(* CODESYS project CodesysElevator.project

Project tree, tasks and I/O mapping:
  CODESYS_Control_Win_V3_x64 : CODESYS Control Win V3 x64, 3S - Smart Software Solutions GmbH, version 3.5.12.30
    application Application
      libraries: BASIC, 3.31 (OSCAT); Util, * (System)
      task VISU_TASK (cyclic, interval 50 ms, priority 31) calls VisuElems.Visu_Prg
      task Task (cyclic, interval t#20ms, priority 1) calls SimulationLogic, main
      Simulation/
        simcomponents/
          visualisation FloorButtons
          visualisation Door
          visualisation Elevator
        SimulationHelpers/
          function block MoveObject [ST]
          function block DoorLogic [ST]
        simlogic/
          program SimIO [ST]
          program SimulationLogic [ST]
        visualisation theLab
      IOs/
        global variables SystemState
        global variables IOs
      control/
        program ElevatorControl [LD]
        program main [ST]
        function block DoorCtrl [SFC]
  libraries: SysTimeCore, 3.5.5.0 (System)
  text list GlobalTextList
*)

// CODESYS_Control_Win_V3_x64/Application/IOs/SystemState
VAR_GLOBAL
	useInputsFromSimulation: BOOL := TRUE;
END_VAR

// CODESYS_Control_Win_V3_x64/Application/IOs/IOs
VAR_GLOBAL
	// inputs
	// Buttons
	ixButtonInElevatorF1: BOOL; // a request in the elevator to go to floor 1
	ixButtonInElevatorF2: BOOL;
	ixButtonInElevatorF3: BOOL;
	ixButtonInElevatorF4: BOOL;
	ixButtonInElevatorCloseDoors: BOOL; // a request to close the door inside the elevator if possible
	ixButtonInElevatorOpenDoors: BOOL; // a request to open the door inside the elevator if possible
	
	// security and sensors
	ixEmergencyStop: BOOL; // Emergency stop is pressed
	ixElevatorAt1: BOOL; // the elevator is at F1 sensor
	ixElevatorAt2: BOOL;
	ixElevatorAt3: BOOL;
	ixElevatorAt4: BOOL;
	ixDoorOpenedF1: BOOL; // the door is fully opened at F1
	ixDoorClosedF1: BOOL; // the door is fully closed at F1
	ixDoorOpenedF2: BOOL;
	ixDoorClosedF2: BOOL;
	ixDoorOpenedF3: BOOL;
	ixDoorClosedF3: BOOL;
	ixDoorOpenedF4: BOOL;
	ixDoorClosedF4: BOOL;

	// outputs
	// lamps
	qxLampInElevatorF1: BOOL;
	qxLampInElevatorF2: BOOL;
	qxLampInElevatorF3: BOOL;
	qxLampInElevatorF4: BOOL;
	qxLampEmergencyStop: BOOL;
	
	qxElevatorGoUp: BOOL;
	qxElevatorGoDown: BOOL;
	qxOpenDoorF1: BOOL; // Opens the door at F1, closes if false
	qxOpenDoorF2: BOOL; // Opens the door at F1, closes if false
	qxOpenDoorF3: BOOL; // Opens the door at F1, closes if false
	qxOpenDoorF4: BOOL; // Opens the door at F1, closes if false
	
END_VAR

// CODESYS_Control_Win_V3_x64/Application/Simulation/simlogic/SimulationLogic
PROGRAM SimulationLogic
VAR
	moveElevator: MoveObject;
	onlyForSimulationElevatorPosY: INT := 0;
	dummyZeroPos: INT := 0;
	elevatorMoving: BOOL;
	
	doorHandleF1: DoorLogic;
	leftPosF1: INT;
	rightPosF1: INT;	
	
	doorHandleF2: DoorLogic;
	leftPosF2: INT;
	rightPosF2: INT;	
	
	doorHandleF3: DoorLogic;
	leftPosF3: INT;
	rightPosF3: INT;	
	
	doorHandleF4: DoorLogic;
	leftPosF4: INT;
	rightPosF4: INT;
	

	
END_VAR


SimIO();



doorHandleF1(leftPos:=leftPosF1, rightPos:= rightPosF1, sensor:= ixElevatorAt1, open := qxOpenDoorF1, close := NOT qxOpenDoorF1);
doorHandleF2(leftPos:=leftPosF2, rightPos:= rightPosF2, sensor:= ixElevatorAt2, open := qxOpenDoorF2, close := NOT qxOpenDoorF2);
doorHandleF3(leftPos:=leftPosF3, rightPos:= rightPosF3, sensor:= ixElevatorAt3, open := qxOpenDoorF3, close := NOT qxOpenDoorF3);
doorHandleF4(leftPos:=leftPosF4, rightPos:= rightPosF4, sensor:= ixElevatorAt4, open := qxOpenDoorF4, close := NOT qxOpenDoorF4);
	

moveElevator(
	moveUP:= SimIO.sim_qxElevatorGoUp, 
	moveDown:= SimIO.sim_qxElevatorGoDown, 
	moveLeft:=FALSE , 
	moveRight:=FALSE , 
	maxX:=0, 
	minX:=0, 
	maxY:=340, 
	minY:=-30, 
	tick:=T#0.03S , 
	x:= dummyZeroPos, 
	y:= onlyForSimulationElevatorPosY );
	
elevatorMoving := moveElevator.isMoving;

END_PROGRAM

// CODESYS_Control_Win_V3_x64/Application/Simulation/simlogic/SimIO
PROGRAM SimIO
VAR
	
	simpleHysteresis: INT := 2;
	posF4: INT := -23;
	posF3: INT := 97;
	posF2: INT := 218;
	posF1: INT := 338;
	
		// for internal simulation use and a way to change bewteen sim and real
	sim_ixButtonAtF1Up: BOOL; 
	sim_ixButtonAtF2Down: BOOL; 
	sim_ixButtonAtF2Up: BOOL;   
	sim_ixButtonAtF3Down: BOOL;
	sim_ixButtonAtF3Up: BOOL;
	sim_ixButtonAtF4Down: BOOL;
	sim_ixButtonInElevatorF1: BOOL; 
	sim_ixButtonInElevatorF2: BOOL;
	sim_ixButtonInElevatorF3: BOOL;
	sim_ixButtonInElevatorF4: BOOL;
	sim_ixButtonInElevatorCloseDoors: BOOL; 
	sim_ixButtonInElevatorOpenDoors: BOOL; 
	
	sim_ixDoorSensorInElevator: BOOL; 
	sim_ixEmergencyStop: BOOL; 
	sim_ixElevatorAt1: BOOL; 
	sim_ixElevatorAt2: BOOL;
	sim_ixElevatorAt3: BOOL;
	sim_ixElevatorAt4: BOOL;
	sim_ixDoorOpenedF1: BOOL; 
	sim_ixDoorClosedF1: BOOL; 
	sim_ixDoorOpenedF2: BOOL;
	sim_ixDoorClosedF2: BOOL;
	sim_ixDoorOpenedF3: BOOL;
	sim_ixDoorClosedF3: BOOL;
	sim_ixDoorOpenedF4: BOOL;
	sim_ixDoorClosedF4: BOOL;

	sim_qxLampAtF1Up: BOOL;
	sim_qxLampAtF2Down: BOOL;
	sim_qxLampAtF2Up: BOOL;
	sim_qxLampAtF3Down: BOOL;
	sim_qxLampAtF3Up: BOOL;
	sim_qxLampAtF4Down: BOOL;
	sim_qxLampInElevatorF1: BOOL;
	sim_qxLampInElevatorF2: BOOL;
	sim_qxLampInElevatorF3: BOOL;
	sim_qxLampInElevatorF4: BOOL;
	sim_qxLampEmergencyStop: BOOL;
	
	sim_qxElevatorGoUp: BOOL;
	sim_qxElevatorGoDown: BOOL;
	sim_qxOpenDoorF1: BOOL; 
	sim_qxOpenDoorF2: BOOL; 
	sim_qxOpenDoorF3: BOOL; 
	sim_qxOpenDoorF4: BOOL; 
END_VAR

// logic

SimIO.sim_ixElevatorAt1 := SimulationLogic.onlyForSimulationElevatorPosY > posF1;
SimIO.sim_ixElevatorAt2 := SimulationLogic.onlyForSimulationElevatorPosY < posF2+simpleHysteresis AND SimulationLogic.onlyForSimulationElevatorPosY > posF2-simpleHysteresis;
SimIO.sim_ixElevatorAt3 := SimulationLogic.onlyForSimulationElevatorPosY < posF3+simpleHysteresis AND SimulationLogic.onlyForSimulationElevatorPosY > posF3-simpleHysteresis;
SimIO.sim_ixElevatorAt4 := SimulationLogic.onlyForSimulationElevatorPosY < posF4;

sim_ixDoorOpenedF1 := SimulationLogic.doorHandleF1.opened;
sim_ixDoorClosedF1 := SimulationLogic.doorHandleF1.closed;
sim_ixDoorOpenedF2 := SimulationLogic.doorHandleF2.opened;
sim_ixDoorClosedF2 := SimulationLogic.doorHandleF2.closed;
sim_ixDoorOpenedF3 := SimulationLogic.doorHandleF3.opened;
sim_ixDoorClosedF3 := SimulationLogic.doorHandleF3.closed;
sim_ixDoorOpenedF4 := SimulationLogic.doorHandleF4.opened;
sim_ixDoorClosedF4 := SimulationLogic.doorHandleF4.closed;


// mapping
IF useInputsFromSimulation THEN
	ixButtonInElevatorF1:=sim_ixButtonInElevatorF1;
	ixButtonInElevatorF2:=sim_ixButtonInElevatorF2;
	ixButtonInElevatorF3:=sim_ixButtonInElevatorF3;
	ixButtonInElevatorF4:=sim_ixButtonInElevatorF4;
	ixButtonInElevatorCloseDoors:=sim_ixButtonInElevatorCloseDoors;
	ixButtonInElevatorOpenDoors:=sim_ixButtonInElevatorOpenDoors;
	
	ixEmergencyStop:=sim_ixEmergencyStop;
	ixElevatorAt1:=sim_ixElevatorAt1;
	ixElevatorAt2:=sim_ixElevatorAt2;
	ixElevatorAt3:=sim_ixElevatorAt3;
	ixElevatorAt4:=sim_ixElevatorAt4;
	ixDoorOpenedF1:=sim_ixDoorOpenedF1;
	ixDoorClosedF1:=sim_ixDoorClosedF1;
	ixDoorOpenedF2:=sim_ixDoorOpenedF2;
	ixDoorClosedF2:=sim_ixDoorClosedF2;
	ixDoorOpenedF3:=sim_ixDoorOpenedF3;
	ixDoorClosedF3:=sim_ixDoorClosedF3;
	ixDoorOpenedF4:=sim_ixDoorOpenedF4;
	ixDoorClosedF4:=sim_ixDoorClosedF4;
END_IF

	sim_qxLampInElevatorF1:=qxLampInElevatorF1;
	sim_qxLampInElevatorF2:=qxLampInElevatorF2;
	sim_qxLampInElevatorF3:=qxLampInElevatorF3;
	sim_qxLampInElevatorF4:=qxLampInElevatorF4;
	sim_qxLampEmergencyStop:=qxLampEmergencyStop;
	
	sim_qxElevatorGoUp:=qxElevatorGoUp;
	sim_qxElevatorGoDown:=qxElevatorGoDown;
	sim_qxOpenDoorF1:=qxOpenDoorF1;
	sim_qxOpenDoorF2:=qxOpenDoorF2;
	sim_qxOpenDoorF3:=qxOpenDoorF3;
	sim_qxOpenDoorF4:=qxOpenDoorF4;

END_PROGRAM

// CODESYS_Control_Win_V3_x64/Application/Simulation/SimulationHelpers/MoveObject
FUNCTION_BLOCK MoveObject
VAR_INPUT
	moveUP: BOOL;
	moveDown: BOOL;
	moveLeft: BOOL;
	moveRight: BOOL;
	maxX: INT;
	minX: INT;
	maxY: INT;
	minY: INT;
	tick: time;
END_VAR
VAR_IN_OUT
	x: INT;
	y: INT;
END_VAR
VAR_OUTPUT
	isMoving: BOOL;
END_VAR
VAR
	pulse: CLK_PULSE;
END_VAR

pulse(
	PT:= tick, 
	N:= 0, 
	RST:= NOT moveUp AND NOT moveDown AND NOT moveLeft AND NOT moveRight , 
	Q=> , 
	CNT=> , 
	RUN=> );
	
IF pulse.Q THEN
	IF moveUP AND NOT moveDown AND y > minY THEN
		y := y-1; 
	ELSIF NOT moveUP AND moveDown AND y < maxY THEN
		y := y+1;
	END_IF
	
	IF moveRight AND NOT moveLeft AND x < maxX THEN
		x := x+1;
	ELSIF NOT moveRight AND moveLeft AND x > minX THEN
		x := x-1;
	END_IF
END_IF

isMoving := moveUP OR moveDown;

END_FUNCTION_BLOCK

// CODESYS_Control_Win_V3_x64/Application/Simulation/SimulationHelpers/DoorLogic
FUNCTION_BLOCK DoorLogic
VAR_INPUT
	open: BOOL;
	close: BOOL;
	sensor: BOOL;
END_VAR
VAR_OUTPUT
	opened: BOOL;
	closed: BOOL;
END_VAR
VAR_IN_OUT
	leftPos: INT;
	rightPos: INT;
END_VAR
VAR
	moveLeft: MoveObject;
	moveRight: MoveObject;
	dummy: INT;
	doOpen: BOOL;
	doClose: BOOL;
END_VAR


opened := leftPos <= -60 AND rightPos >= 60;
closed := leftPos >= 0 AND rightPos <= 0;

doOpen := open AND NOT opened AND NOT close;
doClose := close AND NOT closed AND NOT open;


moveLeft(
	moveUP:= FALSE, 
	moveDown:= FALSE, 
	moveLeft:=doOpen, 
	moveRight:=doClose, 
	maxX:=300, 
	minX:=-300, 
	maxY:=0, 
	minY:=0, 
	tick:=T#0.03S , 
	x:= leftPos, 
	y:= dummy
);

moveRight(
	moveUP:= FALSE, 
	moveDown:= FALSE, 
	moveLeft:=doClose , 
	moveRight:=doOpen , 
	maxX:=300, 
	minX:=-300, 
	maxY:=0, 
	minY:=0, 
	tick:=T#0.03S , 
	x:= rightPos, 
	y:= dummy
);

END_FUNCTION_BLOCK

// CODESYS_Control_Win_V3_x64/Application/control/main
PROGRAM main
VAR
END_VAR

ElevatorControl();

END_PROGRAM

// CODESYS_Control_Win_V3_x64/Application/control/ElevatorControl
PROGRAM ElevatorControl
VAR
	requestF1: BOOL := FALSE;
	requestF2: BOOL := FALSE;
	requestF3: BOOL := FALSE;
	requestF4: BOOL := TRUE;
	r1: BOOL;
	r2: BOOL;
	r3: BOOL;
	r4: BOOL := TRUE;
	up: BOOL := TRUE;
	down: BOOL;
	doorF1: DoorCtrl;
	doorF2: DoorCtrl;
	doorF3: DoorCtrl;
	doorF4: DoorCtrl;
	insane_closing_skills: BOOL := TRUE;
	not_moving: BOOL;
	insane_opening_skills: BOOL;
	going_up: BOOL := TRUE;
	executing1: BOOL;
	executing2: BOOL;
	executing3: BOOL;
	executing4: BOOL;
	executing: BOOL;
	at_stop: BOOL;
	lastF1: BOOL;
	lastF2: BOOL;
	lastF3: BOOL;
	lastF4: BOOL;
END_VAR
VAR // added by the converter: edge detectors and wires of the graphical bodies
    _rt1, _rt2, _rt3, _rt4, _rt5 : R_TRIG;
    _ft1, _ft2, _ft3, _ft4, _ft5, _ft6, _ft7, _ft8, _ft9, _ft10, _ft11, _ft12 : F_TRIG;
END_VAR

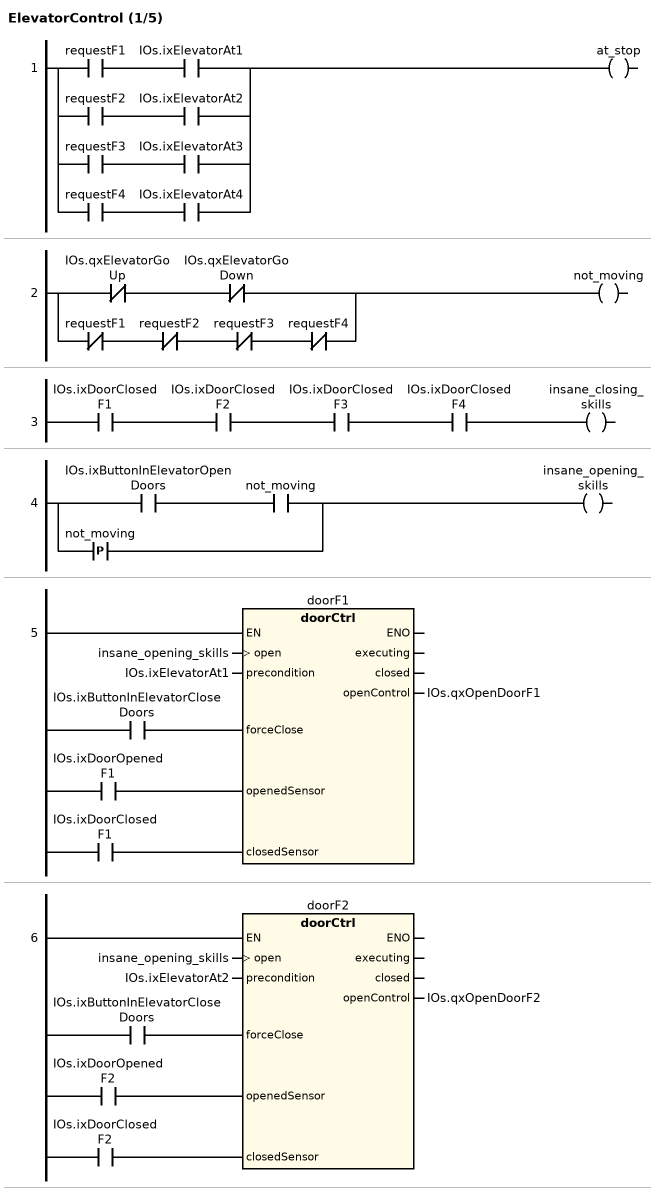
// NETWORK 1
at_stop := requestF1 AND IOs.ixElevatorAt1 OR requestF2 AND IOs.ixElevatorAt2 OR requestF3 AND IOs.ixElevatorAt3 OR requestF4 AND IOs.ixElevatorAt4;

// NETWORK 2
not_moving := NOT IOs.qxElevatorGoUp AND NOT IOs.qxElevatorGoDown OR NOT requestF1 AND NOT requestF2 AND NOT requestF3 AND NOT requestF4;

// NETWORK 3
insane_closing_skills := IOs.ixDoorClosedF1 AND IOs.ixDoorClosedF2 AND IOs.ixDoorClosedF3 AND IOs.ixDoorClosedF4;

// NETWORK 4
_rt1(CLK := not_moving);
insane_opening_skills := IOs.ixButtonInElevatorOpenDoors AND not_moving OR _rt1.Q;

// NETWORK 5
_rt2(CLK := insane_opening_skills);
doorF1(
    open := _rt2.Q,
    precondition := IOs.ixElevatorAt1,
    forceClose := IOs.ixButtonInElevatorCloseDoors,
    openedSensor := IOs.ixDoorOpenedF1,
    closedSensor := IOs.ixDoorClosedF1,
    openControl => IOs.qxOpenDoorF1); // doorCtrl

// NETWORK 6
_rt3(CLK := insane_opening_skills);
doorF2(
    open := _rt3.Q,
    precondition := IOs.ixElevatorAt2,
    forceClose := IOs.ixButtonInElevatorCloseDoors,
    openedSensor := IOs.ixDoorOpenedF2,
    closedSensor := IOs.ixDoorClosedF2,
    openControl => IOs.qxOpenDoorF2); // doorCtrl

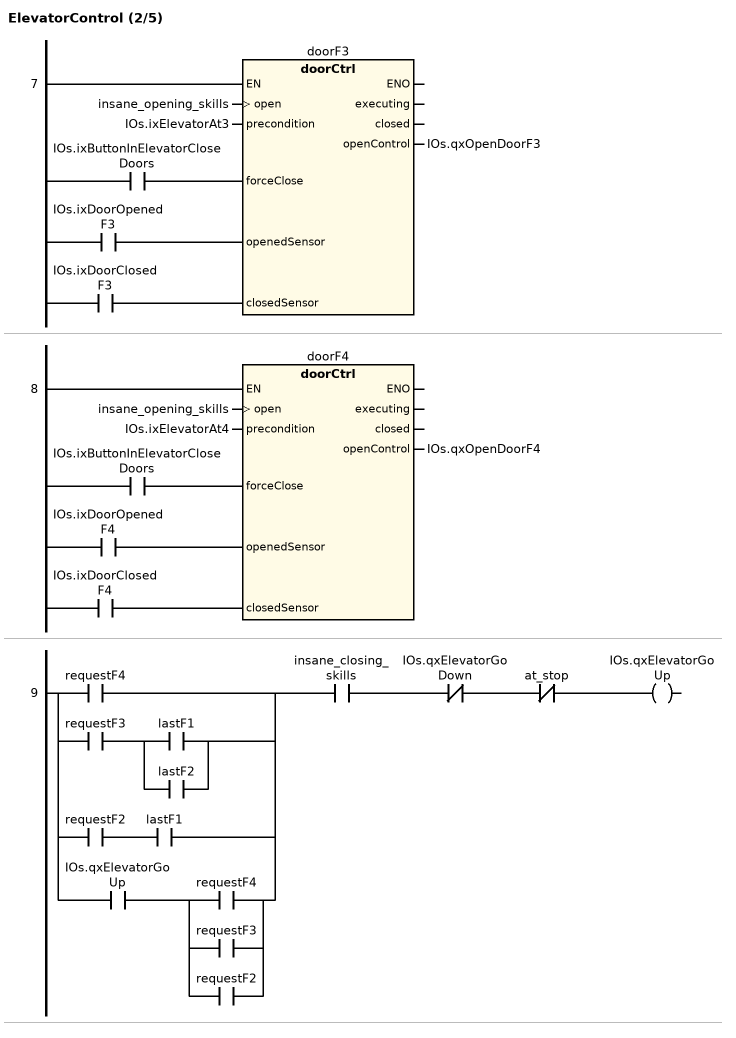
// NETWORK 7
_rt4(CLK := insane_opening_skills);
doorF3(
    open := _rt4.Q,
    precondition := IOs.ixElevatorAt3,
    forceClose := IOs.ixButtonInElevatorCloseDoors,
    openedSensor := IOs.ixDoorOpenedF3,
    closedSensor := IOs.ixDoorClosedF3,
    openControl => IOs.qxOpenDoorF3); // doorCtrl

// NETWORK 8
_rt5(CLK := insane_opening_skills);
doorF4(
    open := _rt5.Q,
    precondition := IOs.ixElevatorAt4,
    forceClose := IOs.ixButtonInElevatorCloseDoors,
    openedSensor := IOs.ixDoorOpenedF4,
    closedSensor := IOs.ixDoorClosedF4,
    openControl => IOs.qxOpenDoorF4); // doorCtrl

// NETWORK 9
IOs.qxElevatorGoUp := (requestF4 OR requestF3 AND (lastF1 OR lastF2) OR requestF2 AND lastF1 OR IOs.qxElevatorGoUp AND (requestF4 OR requestF3 OR requestF2)) AND insane_closing_skills AND NOT IOs.qxElevatorGoDown AND NOT at_stop;

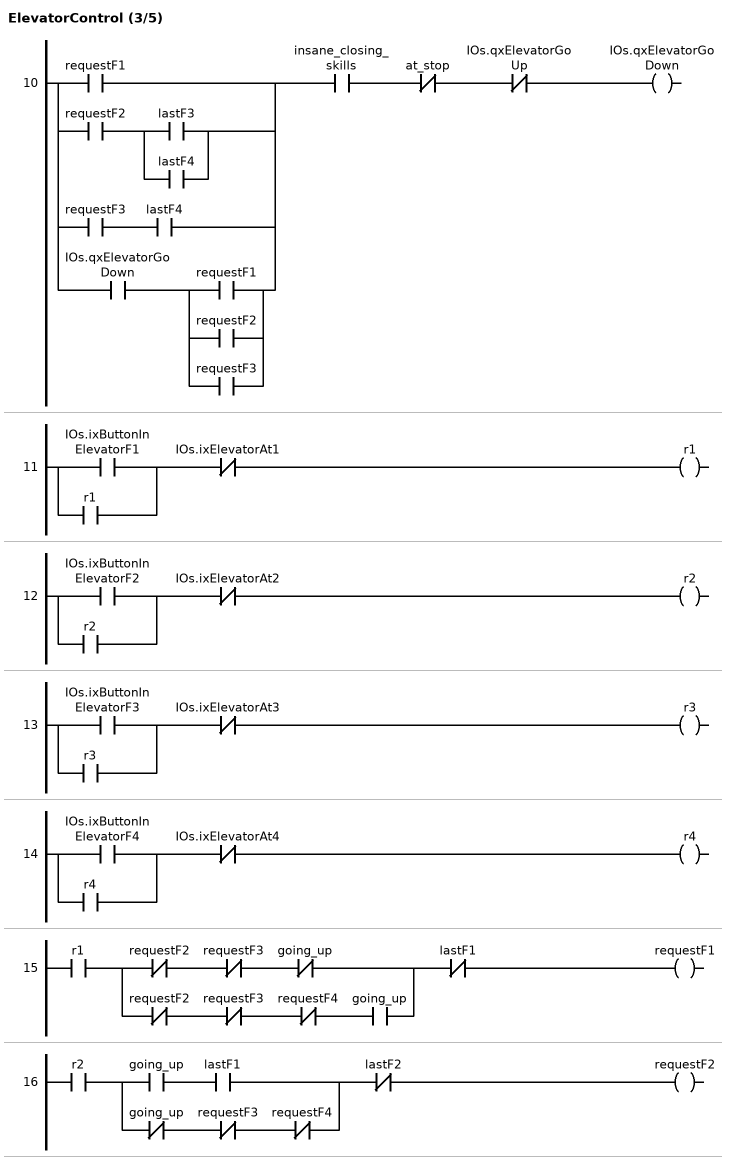
// NETWORK 10
IOs.qxElevatorGoDown := (requestF1 OR requestF2 AND (lastF3 OR lastF4) OR requestF3 AND lastF4 OR IOs.qxElevatorGoDown AND (requestF1 OR requestF2 OR requestF3)) AND insane_closing_skills AND NOT at_stop AND NOT IOs.qxElevatorGoUp;

// NETWORK 11
r1 := (IOs.ixButtonInElevatorF1 OR r1) AND NOT IOs.ixElevatorAt1;

// NETWORK 12
r2 := (IOs.ixButtonInElevatorF2 OR r2) AND NOT IOs.ixElevatorAt2;

// NETWORK 13
r3 := (IOs.ixButtonInElevatorF3 OR r3) AND NOT IOs.ixElevatorAt3;

// NETWORK 14
r4 := (IOs.ixButtonInElevatorF4 OR r4) AND NOT IOs.ixElevatorAt4;

// NETWORK 15
requestF1 := r1 AND (NOT requestF2 AND NOT requestF3 AND NOT going_up OR NOT requestF2 AND NOT requestF3 AND NOT requestF4 AND going_up) AND NOT lastF1;

// NETWORK 16
requestF2 := r2 AND (going_up AND lastF1 OR NOT going_up AND NOT requestF3 AND NOT requestF4) AND NOT lastF2;

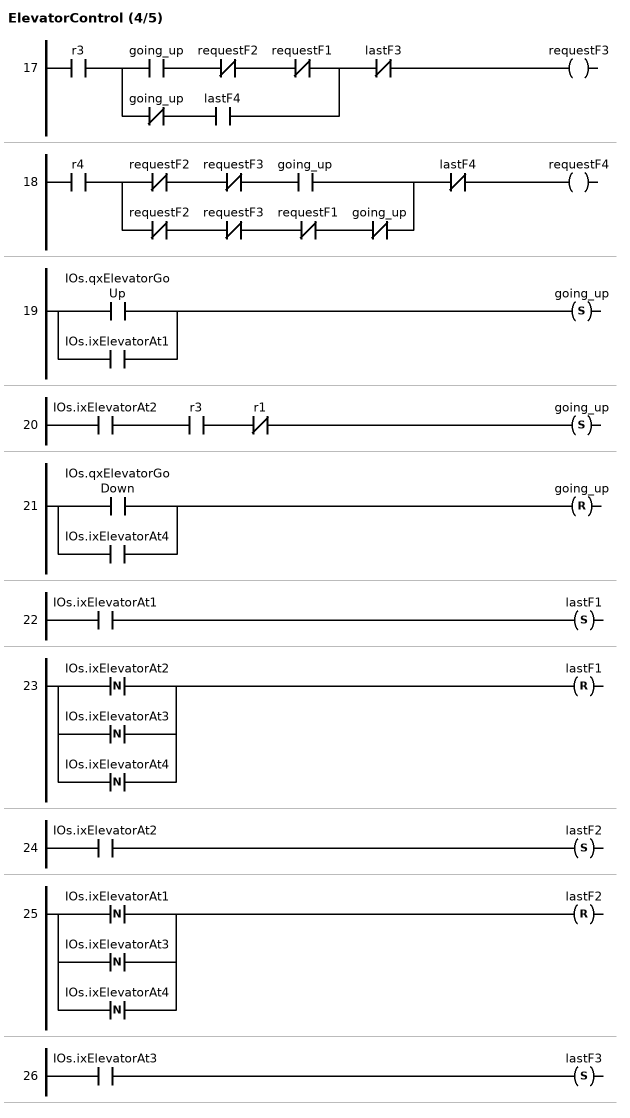
// NETWORK 17
requestF3 := r3 AND (going_up AND NOT requestF2 AND NOT requestF1 OR NOT going_up AND lastF4) AND NOT lastF3;

// NETWORK 18
requestF4 := r4 AND (NOT requestF2 AND NOT requestF3 AND going_up OR NOT requestF2 AND NOT requestF3 AND NOT requestF1 AND NOT going_up) AND NOT lastF4;

// NETWORK 19
going_up S= IOs.qxElevatorGoUp OR IOs.ixElevatorAt1;

// NETWORK 20
going_up S= IOs.ixElevatorAt2 AND r3 AND NOT r1;

// NETWORK 21
going_up R= IOs.qxElevatorGoDown OR IOs.ixElevatorAt4;

// NETWORK 22
lastF1 S= IOs.ixElevatorAt1;

// NETWORK 23
_ft1(CLK := IOs.ixElevatorAt2);
_ft2(CLK := IOs.ixElevatorAt3);
_ft3(CLK := IOs.ixElevatorAt4);
lastF1 R= _ft1.Q OR _ft2.Q OR _ft3.Q;

// NETWORK 24
lastF2 S= IOs.ixElevatorAt2;

// NETWORK 25
_ft4(CLK := IOs.ixElevatorAt1);
_ft5(CLK := IOs.ixElevatorAt3);
_ft6(CLK := IOs.ixElevatorAt4);
lastF2 R= _ft4.Q OR _ft5.Q OR _ft6.Q;

// NETWORK 26
lastF3 S= IOs.ixElevatorAt3;

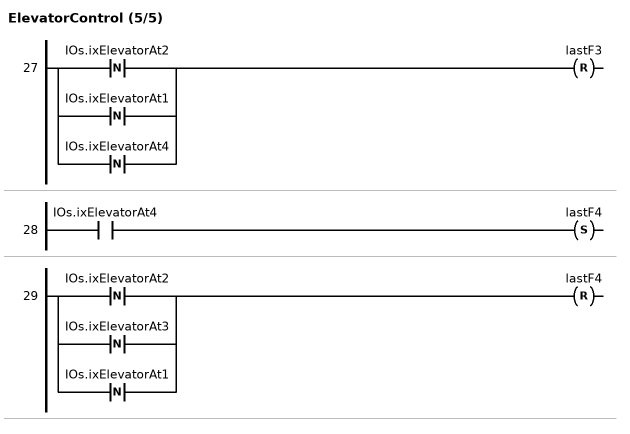
// NETWORK 27
_ft7(CLK := IOs.ixElevatorAt2);
_ft8(CLK := IOs.ixElevatorAt1);
_ft9(CLK := IOs.ixElevatorAt4);
lastF3 R= _ft7.Q OR _ft8.Q OR _ft9.Q;

// NETWORK 28
lastF4 S= IOs.ixElevatorAt4;

// NETWORK 29
_ft10(CLK := IOs.ixElevatorAt2);
_ft11(CLK := IOs.ixElevatorAt3);
_ft12(CLK := IOs.ixElevatorAt1);
lastF4 R= _ft10.Q OR _ft11.Q OR _ft12.Q;

END_PROGRAM

// CODESYS_Control_Win_V3_x64/Application/control/DoorCtrl
FUNCTION_BLOCK DoorCtrl
VAR_INPUT
	open: BOOL;
	precondition: BOOL;
	forceClose: BOOL;
	openedSensor: BOOL;
	closedSensor: BOOL;
END_VAR
VAR_OUTPUT
	executing: BOOL;
	closed: BOOL;
	openControl: BOOL;
END_VAR
VAR
END_VAR

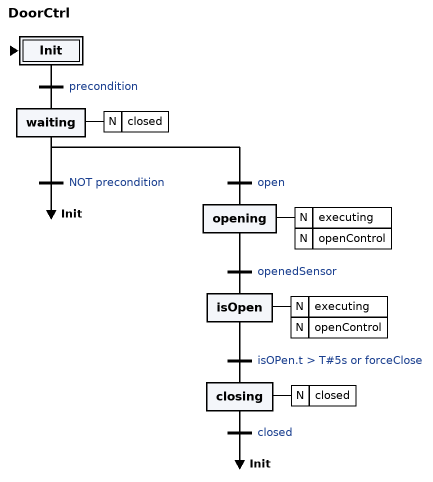
INITIAL_STEP Init:
END_STEP
TRANSITION FROM Init TO waiting
    := precondition;
END_TRANSITION
STEP waiting:
    closed(N);
END_STEP
TRANSITION FROM waiting TO Init
    := NOT precondition;
END_TRANSITION
TRANSITION FROM waiting TO opening
    := open;
END_TRANSITION
STEP opening:
    executing(N);
    openControl(N);
END_STEP
TRANSITION FROM opening TO isOpen
    := openedSensor;
END_TRANSITION
STEP isOpen:
    executing(N);
    openControl(N);
END_STEP
TRANSITION FROM isOpen TO closing
    := isOPen.t > T#5s or forceClose;
END_TRANSITION
STEP closing:
    closed(N);
END_STEP
TRANSITION FROM closing TO Init
    := closed;
END_TRANSITION

END_FUNCTION_BLOCK

// CODESYS_Control_Win_V3_x64/Application/Simulation/simcomponents/FloorButtons
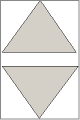
VISUALIZATION FloorButtons  // 80x120
VAR_IN_OUT
	clickUp: BOOL;
	clickDown: BOOL;
	lampUP: BOOL;
	lampDown: BOOL;
END_VAR
    Polygon (2,52) (40,0) (76,52), colour toggle: lampUP
        tap clickUp
    Polygon (2,66) (39,118) (78,66), colour toggle: lampDown
        tap clickDown
END_VISUALIZATION

// CODESYS_Control_Win_V3_x64/Application/Simulation/simcomponents/Door
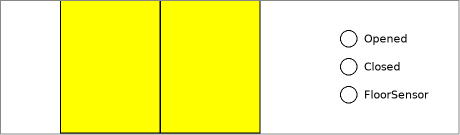
VISUALIZATION Door  // 460x135
VAR_IN_OUT
	opened: BOOL;
	closed: BOOL;
	sensor: BOOL;
	posL: INT;
	posR: INT;
END_VAR
    Rectangle (60,0 100x133)
        p3560616238: posL
    Rectangle (160,0 100x133)
        p3560616238: posR
    Ellipse (340,30 17x17), colour toggle: opened
    Label (361,24 57x30), "Opened"
    Ellipse (340,58 17x17), colour toggle: closed
    Label (361,52 57x30), "Closed"
    Ellipse (340,86 17x17), colour toggle: sensor
    Label (361,80 97x30), "FloorSensor"
END_VISUALIZATION

// CODESYS_Control_Win_V3_x64/Application/Simulation/theLab
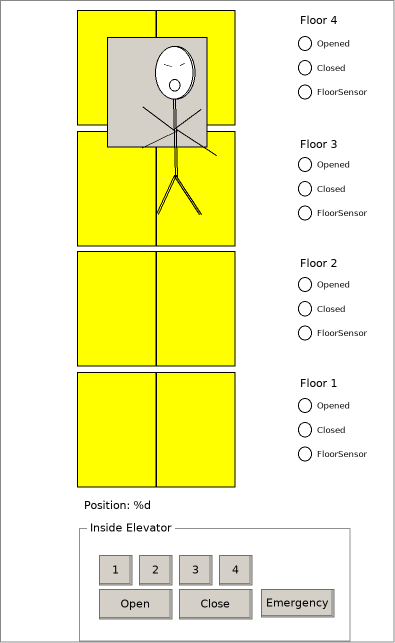
VISUALIZATION theLab  // 395x643
    Frame (30,372 363x117)
        shows Door(opened := SimulationLogic.doorHandleF1.opened, closed := SimulationLogic.doorHandleF1.closed, sensor := SimulationLogic.doorHandleF1.sensor, posL := SimulationLogic.leftPosF1, posR := SimulationLogic.rightPosF1)
    Frame (30,131 363x117)
        shows Door(opened := SimulationLogic.doorHandleF3.opened, closed := SimulationLogic.doorHandleF3.closed, sensor := SimulationLogic.doorHandleF3.sensor, posL := SimulationLogic.leftPosF3, posR := SimulationLogic.rightPosF3)
    Frame (30,251 363x117)
        shows Door(opened := SimulationLogic.doorHandleF2.opened, closed := SimulationLogic.doorHandleF2.closed, sensor := SimulationLogic.doorHandleF2.sensor, posL := SimulationLogic.leftPosF2, posR := SimulationLogic.rightPosF2)
    Frame (30,10 363x117)
        shows Door(opened := SimulationLogic.doorHandleF4.opened, closed := SimulationLogic.doorHandleF4.closed, sensor := SimulationLogic.doorHandleF4.sensor, posL := SimulationLogic.leftPosF4, posR := SimulationLogic.rightPosF4)
    Rectangle (81,494 179x23), "Position: %d", text variable: simulationLogic.onlyForSimulationElevatorPosY
    RoundedRectangle (107,37 100x110)
        p2738717112: SimulationLogic.onlyForSimulationElevatorPosY
    Group (142,46 38x95), invisible if: SimulationLogic.moveElevator.isMoving
        p2738717112: SimulationLogic.onlyForSimulationElevatorPosY
        Ellipse (15,0 38x53)
        Line (61,63)
        Line (33,53) (35,131)
        Line (34,83) (74,109)
        Line (35,85) (0,102)
        Line (34,129) (16,168)
        Line (34,130) (59,168)
        Line (26,39) (43,39)
        Line (23,24) (31,20)
        Line (40,19) (44,23)
    Group (143,46 31x95), invisible if: not SimulationLogic.elevatorMoving
        p2738717112: SimulationLogic.onlyForSimulationElevatorPosY
        Ellipse (12,0 38x53)
        Line (58,63)
        Line (30,53) (32,131)
        Line (31,83) (58,63)
        Line (32,85) (0,61)
        Line (31,129) (13,168)
        Line (31,130) (56,168)
        Line (21,18) (28,20)
        Line (37,19) (41,17)
        Ellipse (26,33 11x12)
    GroupBox (79,520 271x121), "Inside Elevator"
        Button (60,35 33x30), "2", colour toggle: SimIO.sim_qxLampInElevatorF2
            tap SimIO.sim_ixButtonInElevatorF2
        Button (100,35 33x30), "3", colour toggle: SimIO.sim_qxLampInElevatorF3
            tap SimIO.sim_ixButtonInElevatorF3
        Button (140,35 33x30), "4", colour toggle: SimIO.sim_qxLampInElevatorF4
            tap SimIO.sim_ixButtonInElevatorF4
        Button (20,35 33x30), "1", colour toggle: SimIO.sim_qxLampInElevatorF1
            tap SimIO.sim_ixButtonInElevatorF1
        Button (20,69 73x30), "Open"
            tap SimIO.sim_ixButtonInElevatorOpenDoors
        Button (100,69 73x30), "Close"
            tap SimIO.sim_ixButtonInElevatorCloseDoors
        Button (182,69 73x28), "Emergency"
            tap SimIO.sim_ixEmergencyStop
    Rectangle (297,372 56x23), "Floor 1"
    Rectangle (297,252 56x23), "Floor 2"
    Rectangle (297,133 56x23), "Floor 3"
    Rectangle (297,9 56x23), "Floor 4"
END_VISUALIZATION

// CODESYS_Control_Win_V3_x64/Application/Simulation/simcomponents/Elevator
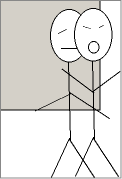
VISUALIZATION Elevator  // 122x179
VAR_IN_OUT
	moving: BOOL;
END_VAR
    RoundedRectangle (0,0 100x110), colour toggle: moving
    Group (35,9 38x95), invisible if: SimulationLogic.moveElevator.isMoving
        Ellipse (15,0 38x53)
        Line (61,63)
        Line (33,53) (35,131)
        Line (34,83) (74,109)
        Line (35,85) (0,102)
        Line (34,129) (16,168)
        Line (34,130) (59,168)
        Line (26,39) (43,39)
        Line (23,24) (31,20)
        Line (40,19) (44,23)
    Group (62,8 31x95), invisible if: not SimulationLogic.elevatorMoving
        Ellipse (12,0 38x53)
        Line (58,63)
        Line (30,53) (32,131)
        Line (31,83) (58,63)
        Line (32,85) (0,61)
        Line (31,129) (13,168)
        Line (31,130) (56,168)
        Line (21,18) (28,20)
        Line (37,19) (41,17)
        Ellipse (26,33 11x12)
END_VISUALIZATION
